// TIA Portal V20 export
DATA_BLOCK "SBK07"   // DB211
// stored: MemoryReserve 100
   VAR
      "X1-0 Gate Cutter Close" : Bool;
      "X2-1 Gate Magazine Close" : Bool;
      "X3-2 Gate Conveyor Close" : Bool;
      "X4-3 reserved" : Bool;
      "X1-4 Gate Cutter Close" : Bool;
      "X2-5 Gate Magazine Close" : Bool;
      "X3-6 Gate Conveyor Close" : Bool;
      "X4-7 reserved" : Bool;
      "X5-0 Gate Cutter Unlock" : Bool;
      "X6-1 Gate Magazine Unlock" : Bool;
      "X7-2 Gate Conveyor Unlock" : Bool;
   END_VAR
BEGIN
END_DATA_BLOCK
